TYPE
  (* Standard: 61131-3; Type: Data Type; Description: Table 12, #5 *)
  (* Version 0.2, 2001-06-14, JHC, Rockwell Automation, Added initial value for MAX_SCALE. *)
  (* Version 0.1, 2001-03-02, JHC, Rockwell Automation, Test for revised Java code generation. *)
  (* Version 0.0, 2000-11-09, JHC, Rockwell Automation *)
  (* Compiler header: package fb.rt.ita; *)
  (* Compiler Java IBM VisualAge 3.0 *)
  (* ASN.1 tag PRIVATE 15 *)
  ANALOG_CHANNEL_CONFIGURATION : STRUCT
    RANGE : ANALOG_SIGNAL_RANGE;
    MIN_SCALE : ANALOG_DATA;
    MAX_SCALE : ANALOG_DATA := 4095;
  END_STRUCT;
END_TYPE
